// TwinCAT 3 PLC project Lift
// ProgramVersion: 3.1.4024.0
// libraries:
//   Tc2_Standard, * (Beckhoff Automation GmbH)
//   Tc2_System, * (Beckhoff Automation GmbH)
//   Tc3_Module, * (Beckhoff Automation GmbH)
//   VisuSymbols,3.5.10.0,System
// project tree:
//   / GlobalTextList.TcGTLO, PlcTask.TcTTO, PlcTask_1.TcTTO, Visualization Manager.TcVMO (not stored)
//   GVLs/ GVL.TcGVL
//   POUs/ CheckIfAtFloor.TcPOU, ledLogic.TcPOU, MAIN.TcPOU
//   VISUs/ Visualization.TcVIS
// real-time tasks:
//   TASK PlcTask: cycle T#10ms, priority 20, ADS port 350
//   TASK PlcTask1: cycle T#10ms, priority 21, ADS port 351

CONFIGURATION Lift
    RESOURCE PLC ON TwinCAT3
        TASK PlcTask(INTERVAL := T#10ms, PRIORITY := 21);
        TASK PlcTask_1(INTERVAL := T#10ms, PRIORITY := 20);
        PROGRAM MAIN WITH PlcTask : MAIN;
        PROGRAM ledLogic WITH PlcTask_1 : ledLogic;
    END_RESOURCE
END_CONFIGURATION

// ---- GVLs/GVL.TcGVL
{attribute 'qualified_only'}
VAR_GLOBAL
	// State cases
	caseInput : INT := 0;
	
	// Instruction string
	instructionString : STRING := 'Initializing lift';

	// General variables
	currentFloor : INT := 0;		// Holds the current floor
	targetFloor : INT := 0;			// The target floor
	liftMoving : BOOL := FALSE;		// Lift is moving
	liftDirection : BOOL := FALSE;	// Lift moving direction (1 is up, 0 is down)
	openDoor : BOOL := FALSE;		// True = open door, False = close door
	liftOperation : BOOL := FALSE;	// True = inside lift, False = outside lift
	
	 // Independent Door Task Control
    doorTask : BOOL := FALSE;         // Activate door task when lift reaches target floor
	
	// Buttons
	callLevel0 : BOOL := FALSE;		// Call base level
	callLevel1 : BOOL := FALSE;		// Call first level
	callLevel2 : BOOL := FALSE;		// Call second level
	setTargetLevel0 : BOOL := FALSE;
	setTargetLevel1 : BOOL := FALSE;
	setTargetLevel2 : BOOL := FALSE;

	// LEDs
	ledLevel0 : BOOL := FALSE;	// Set target floor to base floor
	ledLevel1 : BOOL := FALSE;	// Set target floor to first floor
	ledLevel2 : BOOL := FALSE;	// Set target floor to seocnd floor
	ledLiftMoving : BOOL := FALSE;
	ledDoorsOpen : BOOL := FALSE;
	
	// Time variables
	simulationTime : TON;			// Timer to simulate lift movement
	simulationPace : TIME := T#3S;	// Simulate lift movement (3 seconds)
    doorOpenPace : TIME := T#5S;      // Simulate door open duration (5 seconds)
END_VAR

// ---- POUs/MAIN.TcPOU
PROGRAM MAIN
VAR
	floorOneLamp : BOOL := FALSE;
END_VAR


CASE GVL.caseInput OF
	0: /// Init lift values
		GVL.instructionString := 'Initialising lift';
		GVL.currentFloor := 0;
		GVL.targetFloor := 0;
		GVL.liftMoving := FALSE;
		GVL.openDoor := FALSE;
		
		// Set lift to operating mode
		GVL.caseInput := 1;

	1: /// Wait for outside user input, set targetfloor and LED
		// Update instruction string
		GVL.instructionString := 'Press any of the outside user input';

		// Set target floor to corresponding button call
		IF GVL.callLevel0 THEN
			GVL.targetFloor := 0;
			
			// Set the case input
			GVL.caseInput := 2;
		ELSIF GVL.callLevel1 THEN
			GVL.targetFloor := 1;
			
			// Set the case input
			GVL.caseInput := 2;
		ELSIF GVL.callLevel2 THEN
			GVL.targetFloor := 2;
			
			// Set the case input
			GVL.caseInput := 2;
		END_IF
			
	2: /// Check if lift current floor == target floor, else move lift to correct floor
		// Update instruction string
		GVL.instructionString := 'Checking if current floor == target floor';
		
		// Check if lift is at target floor
		IF CheckIfAtFloor() THEN
			
			// Update instruction string
			GVL.instructionString := 'Arrived at target floor, opening lift doors and waiting for inside user input';
				
			// If floor was called from outside 
			IF GVL.liftOperation = FALSE THEN
				// Open doors
				GVL.openDoor := TRUE;
				
				// Wait for input inside lift
				GVL.caseInput := 5;	
				
			// If floor was called from inside
			ELSIF GVL.liftOperation = TRUE THEN
				// Update instruction string
				GVL.instructionString := 'Arrived at target floor, waiting for user to exis (3s)';

				// Open doors
				GVL.openDoor := TRUE;
				
				// Simulate lift door timer
				GVL.simulationTime(IN := TRUE, PT := GVL.simulationPace);
				
				// Simulate lift door timer
				IF GVL.simulationTime.Q THEN
					// Update instruction string
					GVL.instructionString := 'Closing lift foors and waiting for new outside user input';
					
					// Reset timer and open doors
					GVL.simulationTime(IN := FALSE);
					GVL.openDoor := FALSE;
					
					// Reset liftOperation
					GVL.liftOperation := FALSE;
					
					// Set case to 2 and wait for outside user input
					GVL.caseInput := 1;			
				END_IF
			END_IF
		END_IF
		
	3: /// Move lift downwards
		
		// Update instruction string
		GVL.instructionString := 'Moving lift downwards';
		
		// Set lift direction and move lift
		GVL.liftDirection := TRUE;
		GVL.liftMoving := TRUE;
		
		// Simulate lift timer
		GVL.simulationTime(IN := TRUE, PT := GVL.simulationPace);
		
		IF GVL.simulationTime.Q THEN
			// Reset timer
			GVL.simulationTime(IN := FALSE);	
		
			// Decrease lift level by 1
			GVL.currentFloor := GVL.currentFloor - 1;
			
			// Set case input
			GVL.caseInput := 2;
		END_IF
		
	4: /// Move lift upwards
		// Update instruction string
		GVL.instructionString := 'Moving lift upwards';
		
		//
		GVL.liftDirection := TRUE;
		GVL.liftMoving := TRUE;
		
		// Set lift direction and move lift
		GVL.simulationTime(IN := TRUE, PT := GVL.simulationPace);
		
		IF GVL.simulationTime.Q THEN
			// Reset timer	
			GVL.simulationTime(IN := FALSE);

			// Increase lift level by 1
			GVL.currentFloor := GVL.currentFloor + 1;
			
			// Set case input
			GVL.caseInput := 2;
		END_IF
		
	5: /// Wait for user input inside lift to move
		// Set target floor to corresponding floor, close doors and move lift
		IF GVL.setTargetLevel0 THEN
			GVL.targetFloor := 0;
			GVL.openDoor := FALSE;
			GVL.liftOperation := TRUE;
			GVL.caseInput := 2;
		ELSIF GVL.setTargetLevel1 THEN
			GVL.targetFloor := 1;
			GVL.openDoor := FALSE;
			GVL.liftOperation := TRUE;
			GVL.caseInput := 2;
		ELSIF GVL.setTargetLevel2 THEN
			GVL.targetFloor := 2;
			GVL.openDoor := FALSE;
			GVL.liftOperation := TRUE;
			GVL.caseInput := 2;
		END_IF
END_CASE

END_PROGRAM

// ---- POUs/CheckIfAtFloor.TcPOU
FUNCTION CheckIfAtFloor : BOOL
VAR_INPUT
	
END_VAR
VAR
END_VAR

IF GVL.targetFloor = GVL.currentFloor THEN
	CheckIfAtFloor := TRUE;
	
	// Wait for user input inside lift
//	GVL.liftOperation := TRUE;
	
	// Stop lift movements
	GVL.liftMoving := FALSE;
//	GVL.ledLiftMoving := FALSE;
	
//	// Turn off ledLevels
//	GVL.ledLevel0 := FALSE;
//	GVL.ledLevel1 := FALSE;
//	GVL.ledLevel2 := FALSE;
	
//	// Open the door
//	GVL.openDoor := TRUE;
//	GVL.ledDoorsOpen := TRUE;
	
//	// SInulate lift timer
//	GVL.simulationTime(IN := TRUE, PT := GVL.simulationPace);
	
//	// SInulate lift door timer
//	IF GVL.simulationTime.Q THEN
//		GVL.simulationTime(IN := FALSE);
//		GVL.openDoor := FALSE;
//		GVL.ledDoorsOpen := FALSE;
		
//		GVL.liftOperation := FALSE;
//		// Set case to 2 and wait for outside user input
//		GVL.caseInput := 1;
//	END_IF

	
ELSIF GVL.targetFloor < GVL.currentFloor THEN
	GVL.caseInput := 3;
ELSIF GVL.targetFloor > GVL.currentFloor THEN
	GVL.caseInput := 4;
END_IF

END_FUNCTION

// ---- POUs/ledLogic.TcPOU
PROGRAM ledLogic
VAR
	floorTwoLamp : BOOL := FALSE;
END_VAR

// Turn of leds
IF CheckIfAtFloor() THEN
	IF GVL.liftOperation = FALSE THEN
		// Turn off buttom ledLevels
		GVL.ledLevel0 := FALSE;
		GVL.ledLevel1 := FALSE;
		GVL.ledLevel2 := FALSE;
		GVL.ledDoorsOpen := TRUE;
	END_IF
END_IF

// Turn on door LED
IF GVL.callLevel0 THEN
	GVL.ledLevel0 := TRUE;
//ELSE GVL.ledLevel0 := FALSE;
END_IF

// Turn on door LED
IF GVL.callLevel1 THEN
	GVL.ledLevel1 := TRUE;
//ELSE GVL.ledLevel1 := FALSE;
END_IF

// Turn on door LED
IF GVL.callLevel2 THEN
	GVL.ledLevel2 := TRUE;
//ELSE GVL.ledLevel2 := FALSE;
END_IF

// Turn on door LED
IF GVL.liftMoving THEN
	GVL.ledLiftMoving := TRUE;
ELSE 
	GVL.ledLiftMoving := FALSE;
END_IF

// Turn on door LED
IF GVL.openDoor THEN
	GVL.ledDoorsOpen := TRUE;
ELSE GVL.ledDoorsOpen := FALSE;
END_IF

END_PROGRAM

// ---- GlobalTextList.TcGTLO
TEXTLIST GlobalTextList
  633 = 'Call lift'
  695 = 'Call lift to base floor'
  46 = 'Call lift to first floor'
  697 = 'Call lift to floor 1'
  572 = 'Call lift to floor 2'
  601 = 'Call lift to second floor'
  94 = 'Current floor: %s'
  161 = 'Door is open'
  540 = 'Inside user input'
  512 = 'Instruction: %s'
  416 = 'Lift arrived at floor 1'
  539 = 'Lift arrived at floor 2'
  34 = 'Lift Moving'
  224 = 'Lift moving'
  195 = 'Move lif to level 0'
  399 = 'Move lif to level 1'
  583 = 'Move lif to level 2'
  442 = 'Move lif to targer'
  427 = 'Outside lift call buttons'
  185 = 'Outside user input'
  417 = 'Ready to enter'
  387 = 'Ready to enter (door is open)'
  475 = 'Select floor from inside the lift'
  183 = 'Test'
  731 = 'Test %s'
  11 = 'Test GVL.currentFloor'
END_TEXTLIST

// ---- VISUs/Visualization.TcVIS
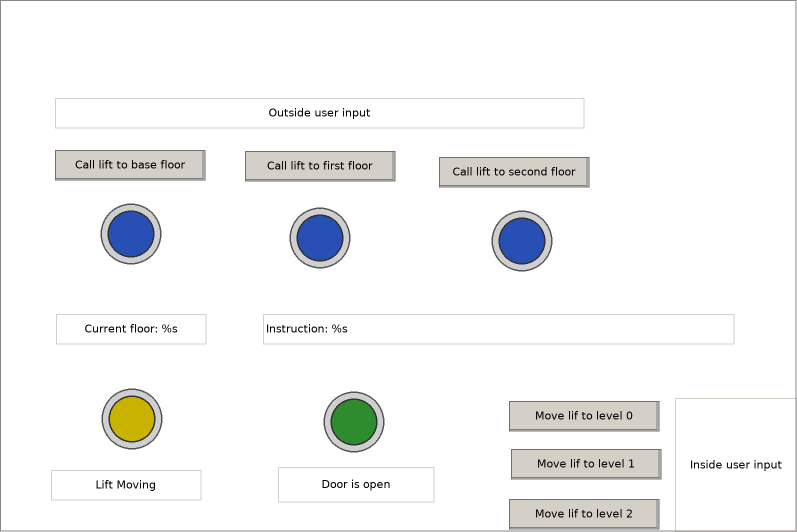
VISUALIZATION Visualization  // 797x532
    Button (55,150 150x30), "Call lift to base floor"
        tap GVL.callLevel0
    Lamp1 (96,199 70x70), variable: GVL.ledLevel0, style: Lamp-Lamp1-Blue
    Lamp1 (319,387 70x70), variable: GVL.ledDoorsOpen, style: Lamp-Lamp1-Green
    Textfield (51,470 150x30), "Lift Moving"
    Button (245,151 150x30), "Call lift to first floor"
        tap GVL.callLevel1
    Lamp1 (285,203 70x70), variable: GVL.ledLevel1, style: Lamp-Lamp1-Blue
    Lamp1 (487,206 70x70), variable: GVL.ledLevel2, style: Lamp-Lamp1-Blue
    Button (509,401 150x30), "Move lif to level 0"
        tap GVL.setTargetLevel0
    Lamp1 (97,384 70x70), tooltip "Lift moving", variable: GVL.ledLiftMoving, style: Lamp-Lamp1-Yellow
    Textfield (278,467 156x35), "Door is open"
    Button (439,157 150x30), "Call lift to second floor"
        tap GVL.callLevel2
    Button (511,449 150x30), "Move lif to level 1"
        tap GVL.setTargetLevel1
    Button (509,499 150x30), "Move lif to level 2"
        tap GVL.setTargetLevel2
    Textfield (56,314 150x30), "Current floor: %s", text variable: GVL.currentFloor
        p4168582468: GVL.currentFloor
    Textfield (263,314 471x30), "Instruction: %s", text variable: GVL.instructionString
        p4168582468: GVL.currentFloor
    Textfield (55,98 529x30), "Outside user input", text variable: GVL.currentFloor
        p4168582468: GVL.currentFloor
    Textfield (675,398 122x134), "Inside user input"
END_VISUALIZATION
